Yaskawa INFORM job: WORKPIECE1.JBI

/JOB
//NAME WORKPIECE1
///FOLDERNAME INNE
//POS
///NPOS 9,9,0,0,0,0
///TOOL 0
///POSTYPE PULSE
///PULSE
C00000=34846,18001,86937,93778,55325,-59342
C00001=34431,-29522,5152,76593,58706,-45262
C00002=35202,-53816,-63523,62971,69519,-31037
C00003=114669,-93784,-99435,114651,-90398,-47027
C00004=113744,-63439,-13119,111243,-76195,-30802
C00005=109933,-121014,-87533,113021,-71100,-39893
C00006=86413,225438,179645,-1854,95162,-11566
C00007=88721,215329,157708,-1846,103518,-10904
C00008=90418,217647,160725,-1786,102890,-10315
BC00000=3493,452410,917391
BC00001=3492,452410,1075223
BC00002=3492,452410,1075223
BC00003=624,80186,893567
BC00004=624,192218,869947
BC00005=9,368120,826334
BC00006=1153,541847,869939
BC00007=24933,423770,872686
BC00008=5,458074,860334
//INST
///DATE 2023/10/04 15:16
///ATTR SC,RW
///GROUP1 RB1,BS1
NOP
'LEFT_SIDE
MOVJ C00000 BC00000 VJ=0.78 PL=0  //POINT1
MOVJ C00001 BC00001 VJ=0.78 PL=0  //POINT2
MOVJ C00002 BC00002 VJ=0.78 PL=0  //POINT3
'BACK_SIDE
MOVJ C00003 BC00003 VJ=0.78 PL=0  //POINT1
MOVJ C00004 BC00004 VJ=0.78 PL=0  //POINT2
MOVJ C00005 BC00005 VJ=0.78 PL=0  //POINT3
'UP_SIDE
MOVJ C00006 BC00006 VJ=0.78 PL=0  //POINT1
MOVJ C00007 BC00007 VJ=0.78 PL=0  //POINT2
MOVJ C00008 BC00008 VJ=0.78 PL=0  //POINT3
END
